TYPE stTableStructx10 :
STRUCT
	b1 : BOOL;
		b2 : BOOL;
			b3 : BOOL;
				b4 : BOOL;
					b5 : BOOL;
						b6 : BOOL;
							b7 : BOOL;
								b8 : BOOL;
									b9 : BOOL;
										b10 : BOOL;
END_STRUCT
END_TYPE

(* stored: Version 1.1.0.1, ProductVersion 3.1.4024.11
   DUT stTableStructx10: Id {84d2b0d5-8048-4032-989f-cd89a19f32f1} *)
